INTERFACE I_BB8Specification

PROPERTY AxisX : I_BasicAxis
GET
END_GET
SET
END_SET
END_PROPERTY

PROPERTY AxisY : I_BasicAxis
GET
END_GET
SET
END_SET
END_PROPERTY

PROPERTY AxisZ : I_BasicAxis
GET
END_GET
SET
END_SET
END_PROPERTY

PROPERTY Config : REFERENCE TO ST_GantryXYZ_Config
GET
END_GET
SET
END_SET
END_PROPERTY

PROPERTY Cylinder : I_Cylinder
GET
END_GET
SET
END_SET
END_PROPERTY

PROPERTY RecipeBuilder : I_RecipeBuilder
GET
END_GET
SET
END_SET
END_PROPERTY

END_INTERFACE

(* stored: Version 1.1.0.1, ProductVersion 3.1.4024.15
   Itf I_BB8Specification: Id {d7ebea93-19fd-4cf9-88f8-8809c3c592f9}
   Property AxisX: Id {4993a6b5-db25-4553-9cb2-07b51c88c577}
   Get Get: Id {522ea5ee-87d4-4fe1-8a51-2790c354af23}
   Set Set: Id {b7ae17ba-0ac9-4c31-93ad-716bc1d77016}
   Property AxisY: Id {6ad5d93f-a2fb-406c-9974-1fbca429a9b8}
   Get Get: Id {ef97a060-0122-4ee5-8991-a29bf266be64}
   Set Set: Id {27ccb336-b0c6-4641-88d0-803685a48b22}
   Property AxisZ: Id {e86eae85-b1a5-453c-a799-0308894c974d}
   Get Get: Id {12ea5ea7-23dd-48d0-8e28-7dae274226fd}
   Set Set: Id {1dc60ee3-7192-45d5-9156-19c0ae6cbb1e}
   Property Config: Id {7be275eb-23e5-4f01-bf6e-fc071cbe44f0}
   Get Get: Id {94c8a7c5-e0c9-491d-85a6-bcea02add430}
   Set Set: Id {7663ee97-65ec-4af7-bc01-7a8bf3fa2b13}
   Property Cylinder: Id {ce125a1d-93e3-4002-8fce-4da998080824}
   Get Get: Id {60d560a9-9bf9-4d2f-acbd-4db7ed3c2b46}
   Set Set: Id {bbf8f8ee-2cf9-4528-8654-cf3c5c11d534}
   Property RecipeBuilder: Id {872801d5-8338-4a69-a743-5f83b587ceb8}
   Get Get: Id {9958ba85-26ba-4191-82c1-9d4bb5d42a94}
   Set Set: Id {b141b14f-8408-4c05-9e89-5c652b07b61a} *)
